PROGRAM Vision
VAR
		BoxLeavesArea	:	BOOL;	// box leaves the filling area and is on the way to vision check
		BoxReadyVision	:	BOOL;	// box ready for vision check
		VisionCheckOk	:	BOOL;	// signal from vision. TRUE if box is OK
		LampBoxOk		:	BOOL;	// signal lamp. Box OK
		LampBoxNok		:	BOOL;	// signal lamp. Box NOK
		StartVision		:	BOOL;	// start vision check
END_VAR
VAR // added by the converter: edge detectors and wires of the graphical bodies
    _w1, _w2 : BOOL;
END_VAR

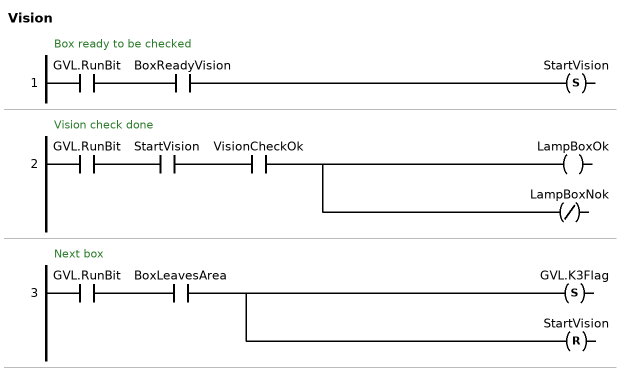
// NETWORK 1
// Box ready to be checked
StartVision S= GVL.RunBit AND BoxReadyVision;

// NETWORK 2
// Vision check done
_w1 := GVL.RunBit AND StartVision AND VisionCheckOk;
LampBoxOk := _w1;
LampBoxNok := NOT _w1;

// NETWORK 3
// Next box
_w2 := GVL.RunBit AND BoxLeavesArea;
GVL.K3Flag S= _w2;
StartVision R= _w2;

END_PROGRAM

(* stored: Version 1.1.0.1, ProductVersion 3.1.4024.15
   POU Vision: Id {723d13ea-1474-4321-8aaf-43d7ae38124f}, SpecialFunc None *)
